TYPE (* logiBUS PI Struct Dual *)
  (* Version 1.0, 2026-05-28, franz *)
  PACKAGE logiBUS::io::PI;
  IMPORT eclipse4diac::core::TypeHash;
  logiBUS_PI_S_Dual : STRUCT
    Up : logiBUS::io::PI::logiBUS_PI_S := (Pin := 255); (* forward, up, right, clockwise *)
    Down : logiBUS::io::PI::logiBUS_PI_S := (Pin := 255); (* backward, down, left, counter-clockwise *)
  END_STRUCT;
END_TYPE
